// TwinCAT 3 PLC project GaragePLC
// ProgramVersion: 3.1.4024.0
// libraries:
//   Tc2_Standard, * (Beckhoff Automation GmbH)
//   Tc2_System, * (Beckhoff Automation GmbH)
//   Tc3_Module, * (Beckhoff Automation GmbH)
//   VisuSymbols,3.5.10.0,System
// project tree:
//   / GlobalTextList.TcGTLO, PlcTask.TcTTO, Task_4.TcTTO, Task_5.TcTTO, VisualizationManager.TcVMO (not stored)
//   GVLs/ Variables.TcGVL
//   POUs/ Door_Control.TcPOU, Light_Control.TcPOU, MAIN.TcPOU, Safety.TcPOU
//   VISUs/ Visualization.TcVIS
// real-time tasks:
//   TASK PlcTask: cycle T#10ms, priority 20, ADS port 350
//   TASK Task 4: cycle T#10ms, priority 21, ADS port 351
//   TASK Task 5: cycle T#10ms, priority 22, ADS port 352

CONFIGURATION GaragePLC
    RESOURCE PLC ON TwinCAT3
        TASK PlcTask(INTERVAL := T#10ms, PRIORITY := 20);
        TASK Task_4(INTERVAL := T#10ms, PRIORITY := 21);
        TASK Task_5(INTERVAL := T#10ms, PRIORITY := 22);
        PROGRAM MAIN WITH PlcTask : MAIN;
        PROGRAM Door_Control WITH Task_4 : Door_Control;
        PROGRAM Light_Control WITH Task_5 : Light_Control;
    END_RESOURCE
END_CONFIGURATION

// ---- GVLs/Variables.TcGVL
VAR_GLOBAL
	Button_Open : BOOL;
	Button_Close : BOOL;
	Sensor_Open : BOOL;
	Sensor_Close : BOOL;
	System_Status : STRING := 'READY';
	Motor_Moving : BOOL;
	Light_Output : BOOL;
	Safety_Sensor :BOOL;
	
END_VAR

// ---- POUs/MAIN.TcPOU
PROGRAM MAIN
VAR
END_VAR

Door_Control();
Light_Control();

END_PROGRAM

// ---- POUs/Door_Control.TcPOU
PROGRAM Door_Control
VAR
	State : INT :=0;
	Safety_Ok : BOOL;
END_VAR

CASE State OF
	0: 	//Idle state 
	Variables.Motor_Moving :=FALSE;
	//Wait for open button
	IF Variables.Button_Open THEN
		State :=10;
	END_IF
	
	10:	// Opening
	Safety_Ok := Safety(Variables.Safety_Sensor); // Check if it is safe
	IF Safety_OK = TRUE THEN
		Variables.Motor_Moving := TRUE; //Tell light task to turn on
		IF Variables.Sensor_Open THEN //Check if door reached the top
			State :=20;
		END_IF
	ELSE 
		State := 0; // Emergency stop
	END_IF
	
	20:	//Opened
	Variables.Motor_Moving :=FALSE;
	IF Variables.Button_Close THEN 	// Wait for close button
		State := 30;
	END_IF
	
	30: //Closing
	Safety_Ok := Safety(Variables.Safety_Sensor);
	IF Safety_Ok = TRUE THEN
		Variables.Motor_Moving := TRUE;
	
	IF Variables.Sensor_Close THEN //Check if door reached the bottom
		State :=0;
	END_IF
	ELSE
		State :=20; // If  there is an obstacle open
	END_IF
END_CASE

END_PROGRAM

// ---- POUs/Safety.TcPOU
FUNCTION Safety : BOOL
VAR_INPUT
	Obstacle : BOOL;
END_VAR
VAR
END_VAR

IF Obstacle =TRUE THEN		// IF there is an obstacle it is not safe
	Safety := FALSE;
	ELSE
		Safety :=TRUE;		// If there is not an obstacle it is safe
END_IF

END_FUNCTION

// ---- POUs/Light_Control.TcPOU
PROGRAM Light_Control
VAR
	Timer : TOF;
END_VAR

Timer(IN :=Variables.Motor_Moving,PT := T#10S); //When the motor stops the light stays on for 10 more seconds
Variables.Light_Output := Timer.Q; //The light stays on if the timer is running

END_PROGRAM

// ---- VISUs/Visualization.TcVIS
VISUALIZATION Visualization  // 2x2
END_VISUALIZATION
